{attribute 'linkalways'} 
{attribute 'no_explicit_call' := 'This FB is a CLASS and must be accessed using methods or properties'}
{attribute 'enable_dynamic_creation'}
FUNCTION_BLOCK FINAL MUL_WORD EXTENDS Node
VAR
	in1 : _WORD(0);
	in2 : _WORD(0);
	out : _WORD(0);
END_VAR

METHOD PUBLIC Clone : I_Node
VAR
	pNode : POINTER TO MUL_WORD;
END_VAR
pNode := __NEW(MUL_WORD);
Clone := pNode^;
END_METHOD

METHOD FB_init : BOOL
VAR_INPUT
	bInitRetains : BOOL; // if TRUE, the retain variables are initialized (warm start / cold start)
	bInCopyCode : BOOL;  // if TRUE, the instance afterwards gets moved into the copy code (online change)
END_VAR
AddInput('in1',THIS^.in1);
AddInput('in2',THIS^.in2);
AddOutput('out', THIS^.out);
END_METHOD

METHOD PROTECTED OnExecute
VAR
END_VAR
out.Value := in1.Value - in2.Value;
END_METHOD

END_FUNCTION_BLOCK

(* stored: Version 1.1.0.1, ProductVersion 3.1.4024.15
   POU MUL_WORD: Id {9807a536-37a1-410a-9a56-85c91af15886}, SpecialFunc None
   Folder Constructor: Id {fdb07be0-111d-458a-9ee3-981f3c554d99}
   Method Clone: Id {4b60d0bc-543f-487c-a33e-71a7b04884d9}
   Method FB_init: Id {ce72ac3d-2579-4bd9-ba65-38c511f2a139}
   Method OnExecute: Id {5cffac1c-1c33-4952-92b7-ad85db20bf55} *)
